TYPE ST_StopSafetyConfig :
STRUCT
    tTimeout : TIME;
END_STRUCT
END_TYPE

(* stored: Version 1.1.0.1, ProductVersion 3.1.4026.20
   DUT ST_StopSafetyConfig: Id {38f6d86f-ac09-4196-97c2-0dc1a77a4812} *)
